% RSLogix 500 project I2P-JOB-22 DUNCAN_SUTTON.RSS, saved by version 10.00.00.00 %
PROJECT "ML01A"    % processor: Bul.1763 MicroLogix 1100 Series B %

PROGRAM FILES
  LAD 2   9 rungs

DATA FILES
  O0 OUTPUT  4 elements
  I1 INPUT  6 elements
  S2 STATUS  66 elements
  B3 BINARY  1 elements
  T4 TIMER  1 elements
  C5 COUNTER  2 elements
  R6 CONTROL  1 elements
  N7 INTEGER  1 elements
  F8 FLOAT  1 elements

LADDER 2
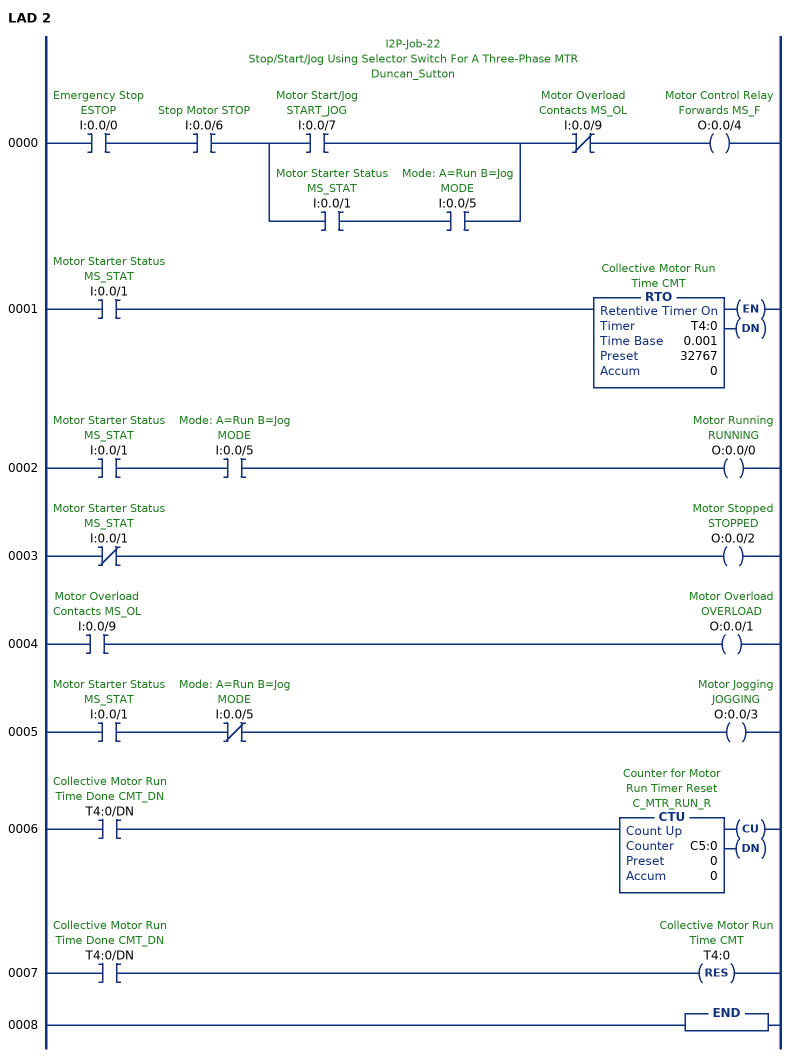
% Rung: 0 %
% I2P-Job-22
% Stop/Start/Jog Using Selector Switch For A Three-Phase MTR
% Duncan_Sutton %
SOR XIC I:0.0/0 XIC I:0.0/6 BST XIC I:0.0/7 NXB XIC I:0.0/1 XIC I:0.0/5 BND XIO I:0.0/9 OTE O:0.0/4 EOR
%   I:0.0/0  ESTOP  "Emergency Stop" %
%   I:0.0/6  STOP  "Stop Motor" %
%   I:0.0/7  START_JOG  "Motor Start/Jog" %
%   I:0.0/1  MS_STAT  "Motor Starter Status" %
%   I:0.0/5  MODE  "Mode: A=Run B=Jog" %
%   I:0.0/9  MS_OL  "Motor Overload Contacts" %
%   O:0.0/4  MS_F  "Motor Control Relay Forwards" %
% Rung: 1 %
SOR XIC I:0.0/1 RTO T4:0 0.001 32767 0 EOR
%   I:0.0/1  MS_STAT  "Motor Starter Status" %
%   T4:0  CMT  "Collective Motor Run Time" %
% Rung: 2 %
SOR XIC I:0.0/1 XIC I:0.0/5 OTE O:0.0/0 EOR
%   I:0.0/1  MS_STAT  "Motor Starter Status" %
%   I:0.0/5  MODE  "Mode: A=Run B=Jog" %
%   O:0.0/0  RUNNING  "Motor Running" %
% Rung: 3 %
SOR XIO I:0.0/1 OTE O:0.0/2 EOR
%   I:0.0/1  MS_STAT  "Motor Starter Status" %
%   O:0.0/2  STOPPED  "Motor Stopped" %
% Rung: 4 %
SOR XIC I:0.0/9 OTE O:0.0/1 EOR
%   I:0.0/9  MS_OL  "Motor Overload Contacts" %
%   O:0.0/1  OVERLOAD  "Motor Overload" %
% Rung: 5 %
SOR XIC I:0.0/1 XIO I:0.0/5 OTE O:0.0/3 EOR
%   I:0.0/1  MS_STAT  "Motor Starter Status" %
%   I:0.0/5  MODE  "Mode: A=Run B=Jog" %
%   O:0.0/3  JOGGING  "Motor Jogging" %
% Rung: 6 %
SOR XIC T4:0/DN CTU C5:0 0 0 EOR
%   T4:0/DN  CMT_DN  "Collective Motor Run Time Done" %
%   C5:0  C_MTR_RUN_R  "Counter for Motor Run Timer Reset" %
% Rung: 7 %
SOR XIC T4:0/DN RES T4:0 EOR
%   T4:0/DN  CMT_DN  "Collective Motor Run Time Done" %
%   T4:0  CMT  "Collective Motor Run Time" %
% Rung: 8 %
SOR END EOR

OTHER DOCUMENTED ADDRESSES
  B3:0/0  B_ESTOP  "B_Estop"
  B3:0/1  B_FWD  "FWD Memory"
  B3:0/2  B_REV  "Reverse Memory"
  B3:0/3  LAST_FWD  "Memory Direction Foward"
  B3:0/4  LAST_REV  "Memory Direction Reverse"
  C5:1  C_MTR_T  "Collective Motor Run Time Counter"
  I:0.0/2  DIR_STAT  "Motor Direction Control Status"
  I:0.0/3  MODE_ON  "Valve Mode ON"
  I:0.0/4  MODE_AUTO  "Valve Mode Auto"
  I:0.0/8  JOG  "JOG Motor"
  I:0.1  MS
  O:0.0/5  CR_2  "Direction Control Relay"
  T4:0.ACC/0  T4
  T4:0.PRE  OVERCLOCK  "Collective Motor OverClock"

DATA TABLE (non-zero values as saved)
DATA B3
% B3:0 % 0X0001
DATA T4
% .PRE .ACC %
% T4:0 % 32767 0
